{attribute addProperty BoxType "EL3681-0000-0021"}
{attribute addProperty Id "SettingsAT %I*Settings_7AA6B313162"}
{attribute addProperty CRC "3751299124"}
{attribute addProperty SizeInBites "16"}
{attribute addProperty SizeInBytes "2"}
TYPE SAI_Feedback_DF984834 :
STRUCT
	{attribute addProperty Name "Settings"}
	Settings AT %I* : Settings_7AA6B313;
END_STRUCT
END_TYPE

(* stored: Version 1.2.0.0, ProductVersion 3.1.4024.9
   DUT SAI_Feedback_DF984834: Id {f6260838-72ab-4dc3-92c6-81b1fabce191} *)
